{attribute 'GeneratedUsingTerminal: EL2521-0124-0016'}
{attribute addProperty BoxType "EL2521-0124-0016"}
{attribute addProperty Id "Enable_PLSAT %Q*BOOL1OutputAT %Q*BOOL1Switch_on_valueAT %Q*UINT2Switch_off_valueAT %Q*UINT2"}
{attribute addProperty CRC "3700533176"}
{attribute addProperty Size "6"}
TYPE PLS_Control_compact_DC91A7B8 :
STRUCT
	{attribute addProperty Name "Enable_PLS"}
	Enable_PLS AT %Q* : BOOL;
	{attribute addProperty Name "Output"}
	Output AT %Q* : BOOL;
	{attribute addProperty Name "Switch_on_value"}
	Switch_on_value AT %Q* : UINT;
	{attribute addProperty Name "Switch_off_value"}
	Switch_off_value AT %Q* : UINT;
END_STRUCT
END_TYPE

(* stored: Version 1.2.0.0, ProductVersion 3.1.4024.9
   DUT PLS_Control_compact_DC91A7B8: Id {da75a213-fa18-4795-82ab-13f157197248} *)
